FUNCTION_BLOCK L5_Panel
VAR_INPUT
	dr								: REFERENCE TO L1_Director;

	mdF1Producir					: BOOL := TRUE;
	//mdF6Probar						: BOOL;
	mdF5Funcion						: BOOL;
	mdF4Planta						: BOOL;

	hwAS_AvisadorSonoro		AT %Q*	: BOOL; 
	hwLA_LamparaAlarma		AT %Q*	: BOOL; 
	//hwDPO_DesconectaPO		AT %Q*	: BOOL; 	
	hwLM_LamparaMarcha		AT %Q*	: BOOL;
	hwLS_LamparaStop		AT %Q*	: BOOL;

	swF0_Empezar					: BOOL;
	swF1_Producir					: BOOL := TRUE;
	swF2_Preparar					: BOOL := TRUE;
	swF3_Finalizar					: BOOL := TRUE;
	swF6_Probar						: BOOL;
	
	swF4_Planta						: BOOL; 
	swMensaje						: STRING(255) :='';
END_VAR

VAR
	hwPE_Seta					AT %I*	: BOOL;
	swPE_Seta							: BOOL;
	
	hwPOC_PulsadorReset			AT %I*	: BOOL; // POC Botón azul está pulsado (PO Conectada)
	swPOC_PulsadorReset					: BOOL; 
	
	hwPM_PulsadorMarcha			AT %I*	: BOOL; // PM - Pulsador de marcha (verde)
	swPM_PulsadorMarcha					: BOOL;
	fpPM_PulsadorMarcha					: R_TRIG;
	clPM_PulsadorMarcha					: TON;
	
	
	hwPS_PulsadorStop			AT %I*	: BOOL := TRUE; // PS - Pulsador de parada (rojo)
	swPS_PulsadorStop					: BOOL := TRUE; 
	fnPS_PulsadorStop					: F_TRIG; 
	
	hwSM_SelecAutoManual	 	AT %I*	: BOOL; // SM - Selector modo auto/man
	swSM_SelecAutoManual	 			: BOOL; 	

END_VAR


VAR_OUTPUT
	// consignas del panel, resultado de integrar la información que viene del hardware, el estado GEMMA, los temporizadores y flancos, y la interfaz de usuario		
	swF4_Avanza						: BOOL := FALSE;
 	swF4_Retroc						: BOOL := FALSE;	
	
	swF5_Alimentar					: BOOL;
	fpF5_Alimentar					: R_TRIG;  // cuando se pulsa alimentar hay que quitar cargar
	swF5_Situar						: BOOL;
	swF5_Transferir					: BOOL;
	fpF5_Transferir					: R_TRIG; // cuando se pulsa transferir hay que quitar descargar
	swF5_Cargar						: BOOL;
	fpF5_Cargar						: R_TRIG; // cuando se pulsa cargar hay que quitar girar y alimentar
	swF5_Evacuar					: BOOL;
	fpF5_Evacuar					: R_TRIG; // cuando se pulsa evacuar hay que quitar girar
	swF5_Descargar					: BOOL;
	fpF5_Descargar					: R_TRIG; // cuando se pulsa descargar hay que quitar girar y transferir
	swF5_Medir						: BOOL;
	fpF5_Medir						: R_TRIG; // cuano se pulsa medir hay que quitar girar
	swF5_Claridad					: BOOL;
	swF5_Material					: BOOL;
	swF5_Girar						: BOOL;
	fpF5_Girar						: R_TRIG; // cuando se pulsa girar hay que quitar medir, cargar, descargar y evacuar
	swF5_Ejecutar					: BOOL;
	swF5_Ack						: BOOL;
	
END_VAR

VAR
	gmModeName		: STRING 	:= 'Mode A6';
	gmModeDescr		: STRING 	:= 'Inicializando';	
	
//	ttPE_Seta						: STRING := '';

	swA2_FinCiclo					: BOOL;
	swA3_Estado						: BOOL;
	swA6_Inicializar				: BOOL;

	//swF2_Preparar					: BOOL;
	//swF3_Finalizar				: BOOL;	
	//ttF4_Planta						: STRING :='';
	//enF6_Probar						: BOOL;
	//swF6_Probar						: BOOL;
END_VAR

METHOD ProcessCycle : BOOL
VAR_INPUT
	dr				: REFEREnce to L1_Director;
	gmModeActual	: L1_GEMMA;
	tmReinicio 		: TIME; // = dr.tmTiempoReinicio
END_VAR
clPM_PulsadorMarcha(IN:=hwPM_PulsadorMarcha OR  swPM_PulsadorMarcha, PT:=T#1S);
fpPM_PulsadorMarcha(CLK:=hwPM_PulsadorMarcha OR  swPM_PulsadorMarcha);
fnPS_PulsadorStop  (CLK:=hwPS_PulsadorStop   AND swPS_PulsadorStop);

IF hwPE_Seta OR swPE_Seta THEN
	dr.cnD1_Emergencia 				:= TRUE;
	dr.cnA6_Inicializar 			:= FALSE;
	dr.cnA3_Estado					:= FALSE; 
	dr.cnF0_Empezar					:= FALSE;
	dr.cnF4_Planta					:= FALSE; // CON LA SETA NO SE PUEDE ENTRAR EN MODO F4
	dr.cnF5_Funcion					:= FALSE; // CON LA SETA NO SE PUEDE ENTRAR EN MODO F5
	swMensaje 						:= 'Parada de emergencia. Desactive la seta y pulse Reset';

ELSIF dr.cnD1_Emergencia AND NOT (hwPE_Seta OR swPE_Seta) THEN	
	dr.cnD1_Emergencia 				:= FALSE;
	dr.cnA6_Inicializar 			:= TRUE;
	swMensaje 						:= 'Inicializando...';

ELSIF dr.cnA6_Inicializar AND dr.IC THEN
	dr.cnA6_Inicializar				:= FALSE;

ELSIF clPM_PulsadorMarcha.Q THEN			// 1o salta el empezar, si tardas más de 1s luego salta la parada
	dr.cnA3_Estado					:= TRUE;
	dr.cnF0_Empezar					:= FALSE;
	
ELSIF dr.cnF1_Producir AND fnPS_PulsadorStop.Q THEN
	dr.cnA2_FinCiclo				:= TRUE;
	
ELSIF dr.cnA3_Estado AND dr.gmModeActual=L1_GEMMA.A4ParadaObtenida THEN
	dr.cnA3_Estado 					:= FALSE;

ELSIF fpPM_PulsadorMarcha.Q THEN
	dr.cnF0_Empezar 				:= TRUE;
	
ELSIF gmModeActual=L1_GEMMA.A1ParadaInicial THEN
	dr.cnF1_Producir			:= swF1_Producir AND NOT swF6_Probar;
	dr.cnF2_Preparar 			:= swF2_Preparar AND NOT swF6_Probar;
	dr.cnF3_Finalizar			:= swF3_Finalizar AND NOT swF6_Probar;
	dr.cnF6_Probar				:= swF6_Probar AND NOT (swF1_Producir OR swF2_Preparar OR swF3_Finalizar);

ELSIF mdF1Producir AND NOT dr.cnF1_Producir THEN								
	mdF1Producir				:= TRUE;
	mdF4Planta					:= FALSE;
	mdF5Funcion					:= FALSE;
	dr.cnF1_Producir			:= TRUE;
	dr.cnF4_Planta				:= FALSE;	
	dr.cnF5_Funcion				:= FALSE;
	swMensaje					:= 'Modo producción activado';
			
//	dr.cnF1_Producir			:= swF1_Producir AND NOT swF6_Probar;
	//dr.cnF2_Preparar 			:= swF2_Preparar AND NOT swF6_Probar;
	//dr.cnF3_Finalizar			:= swF3_Finalizar AND NOT swF6_Probar;
	//dr.cnF6_Probar				:= swF6_Probar AND NOT (swF1_Producir OR swF2_Preparar OR swF3_Finalizar);		

ELSIF (hwSM_SelecAutoManual OR swSM_SelecAutoManual) AND NOT DR.cnF4_Planta THEN // paso al modo F4
	mdF1Producir				:= FALSE;
	mdF4Planta					:= TRUE;
	mdF5Funcion					:= FALSE;
	dr.cnF1_Producir			:= FALSE;
	dr.cnF4_Planta				:= TRUE;	
	dr.cnF5_Funcion				:= FALSE;
	swMensaje					:= 'Modo mando directo activado';

ELSIF gmModeActual=L1_GEMMA.F4VerificacionSinOrden AND 
	NOT (hwSM_SelecAutoManual OR swSM_SelecAutoManual) THEN
	dr.cnF4_Planta				:= FALSE;
	swSM_SelecAutoManual		:= FALSE;
	swMensaje					:= 'Modo F4 desactivado';

ELSIF mdF5Funcion AND NOT dr.cnF5_Funcion THEN
	mdF1Producir				:= FALSE;
	mdF4Planta					:= FALSE;
	mdF5Funcion					:= TRUE;
	dr.cnF1_Producir			:= FALSE;
	dr.cnF4_Planta				:= FALSE;	
	dr.cnF5_Funcion				:= TRUE;
	swMensaje					:= 'Modo función activado';

END_IF
            




IF gmModeActual=L1_GEMMA.F5VerificacionOrdenada THEN
	
	//IF NOT mdF5Funcion OR NOT mdF5Funcion OR hwSM_SelecAutoManual OR swSM_SelecAutoManual THEN
	//	dr.cnF5_Funcion				:= FALSE;
	//	mdF5Funcion					:= FALSE;
	//	IF hwSM_SelecAutoManual OR swSM_SelecAutoManual THEN
	//		dr.cnF4_Planta			:= TRUE;
	//		swMensaje					:= 'Modo F4 activado';
	//	ELSE
		//	swMensaje					:= 'Modo F5 desactivado';			
		//END_IF
		
	//ELSE
	fpF5_Alimentar				(CLK := swF5_Alimentar);
	fpF5_Cargar					(CLK := swF5_Cargar);
	fpF5_Medir					(CLK := swF5_Medir);
	fpF5_Evacuar				(CLK := swF5_Evacuar);
	fpF5_Descargar				(CLK := swF5_Descargar);
	fpF5_Girar					(CLK :=swF5_Girar);
	fpF5_Transferir				(CLK :=swF5_Transferir);
	IF fpF5_Alimentar.Q AND swF5_Cargar THEN
		swF5_Cargar				:= FALSE; 
		swMensaje				:= 'No se puede cargar si se alimenta';
	ELSIF fpF5_Cargar.Q AND (swF5_Alimentar OR swF5_Girar)THEN
		swF5_Alimentar			:= FALSE; 
		swF5_Girar				:= FALSE;
		swMensaje				:= 'No se puede alimentar ni girar si se carga';		
	ELSIF fpF5_Medir.Q AND swF5_Girar THEN
		swF5_Girar				:= FALSE; 
		swMensaje				:= 'No se puede girar si se mide';
	ELSIF fpF5_Evacuar.Q AND swF5_Girar THEN	
		swF5_Girar				:= FALSE; 
		swMensaje				:= 'No se puede girar si se evacúa';
	ELSIF fpF5_Descargar.Q AND (swF5_Girar OR swF5_Transferir) THEN
		swF5_Girar				:= FALSE; 
		swF5_Transferir			:= FALSE;
		swMensaje				:= 'No se puede girar ni transferir si se descarga';
	ELSIF fpF5_Girar.Q AND (swF5_Cargar OR swF5_Medir OR swF5_Evacuar OR swF5_Descargar) THEN
		swF5_Cargar				:= FALSE;
		swF5_Medir				:= FALSE;
		swF5_Evacuar			:= FALSE;
		swF5_Descargar			:= FALSE;
		swMensaje				:= 'No se puede cargar, medir, evacuar ni descargar si se gira';
	ELSIF fpF5_Transferir.Q AND swF5_Descargar THEN
		swF5_Descargar			:= FALSE; 
		swMensaje				:= 'No se puede descargar si se transfiere';
	END_IF		
END_IF
UpdateUI(gmMode := dr.gmModeActual);

 
//ELSE
	(*

ttPE_Seta := 'Pulsar la seta o el botón para parada de emergencia';	
ttF4_Planta := 'Mandos directos desactivados';
FP_PM(CLk := hwPM_PulsadorMarcha);

dr.cnA1_ParadaIni := FALSE;
	dr.cnA6_Inicializar := FALSE; 
	dr.cnF4_Planta 		:= FALSE;
	dr.cnF5_Funcion 	:= FALSE;
	dr.cnF6_Probar 		:= FALSE;
	dr.cnF1_Producir	:= FALSE;

//----------------------------------------------------------------- Consiga cnD1_Emergencia
dr.cnD1_Emergencia := hwPE_Seta OR swPE_Seta; 
IF dr.cnD1_Emergencia THEN
	IF hwPE_Seta THEN
		IF swPE_Seta THEN
			ttPE_Seta := 'Desarmar la seta y desactivar el botón para reinicializar';
		ELSE
			ttPE_Seta := 'Desarmar la seta para reinicializar';		
		END_IF
	ELSE
		IF swPE_Seta THEN
			ttPE_Seta := 'Desactivar el botón para reinicializar';
		END_IF
	END_IF

//----------------------------------------------------------------- Consigna A6_Inicializar
ELSIF swA6_Inicializar THEN //  OR TmpReinicio.Q);
	// TmpReinicio(IN := hwPM_PulsadorMarcha AND NOT hwPS_PulsadorStop, PT:= tmReinicio);
	dr.cnA6_Inicializar := TRUE; 
	//mdF1Producir := FALSE;
	//mdF4Planta := FALSE;
	//mdF5Funcion := FALSE;
	//mdF6Probar := FALSE;
 
	
//----------------------------------------------------------------- Modo F4_Planta
ELSIF (hwSM_SelecAutoManual OR mdF4Planta) THEN 
	//mdF1Producir 	:= FALSE;
	dr.cnF4_Planta 	:= TRUE;
	//dr.cnF5_Funcion := TRUE;
	//mdF5Funcion 	:= FALSE;
	//mdF6Probar 		:= FALSE;
	IF hwSM_SelecAutoManual AND swF4_Planta THEN
		ttF4_Planta := 'Mandos directos ativados desde panel físico y visualización';
	ELSIF hwSM_SelecAutoManual THEN	
		ttF4_Planta := 'Mandos directos ativados desde panel físico';
	ELSIF swF4_Planta THEN
		ttF4_Planta := 'Mandos directos ativados desde visualización';
	END_IF	

	
	

//----------------------------------------------------------------- F5_Funcion
ELSIF mdF5Funcion THEN  
	//mdF1Producir 	:= FALSE;
	//mdF4Planta 		:= FALSE;
	dr.cnF5_Funcion := TRUE;
	//mdF6Probar 		:= FALSE;

	IF swF5_Girar AND (swF5_Cargar OR swF5_Evacuar OR swF5_Descargar OR swF5_Medir) THEN 
		//swF5_Girar := FALSE;
		swF5_Cargar := FALSE;
		swF5_Evacuar := FALSE;
		swF5_Descargar := FALSE;
		swF5_Medir := FALSE;
		swMensaje := 'No se puede girar a la vez que cargar, evacuar, descargar o medir por riesgo de avería';
	END_IF
	IF swF5_Alimentar AND swF5_Cargar THEN // funciones incompatibles
		swF5_Cargar := FALSE;
		swMensaje := 'No se puede cargar a la vez que alimentar por riesgo de avería';
	END_IF
	IF swF5_Transferir AND swF5_Descargar THEN
		swF5_Transferir := FALSE;
		swMensaje := 'No se puede descargar a la vez que transferer por riesgo de avería';
	END_IF


	
//----------------------------------------------------------------- F6_Probar
ELSIF mdF6Probar THEN  
	//mdF1Producir	:= FALSE;
	//mdF4Planta 		:= FALSE;
	//mdF5Funcion 	:= FALSE;
	dr.cnA1_ParadaIni := NOT dr.cnF0_Empezar;
	dr.cnF6_Probar 	:= TRUE;
	IF (swF0_Empezar OR FP_PM.Q) THEN
		dr.cnF0_Empezar := TRUE;
	END_IF

	
//----------------------------------------------------------------- F1_Producir
ELSIF (mdF1Producir OR FP_PM.Q) THEN
	dr.cnF1_Producir:= TRUE;

	IF (swF0_Empezar OR FP_PM.Q) THEN
		dr.cnF0_Empezar := TRUE;
	END_IF
	//dr.cnF0_Empezar := (swF0_Empezar OR FP_PM.Q);  
	dr.cnA1_ParadaIni := NOT dr.cnF0_Empezar;
	//mdF4Planta 		:= FALSE;
	//mdF5Funcion 	:= FALSE;
	//mdF6Probar	 	:= FALSE;

	dr.cnA2_FinCiclo:= (swA2_FinCiclo OR hwPS_PulsadorStop); // enA2_FinCiclo AND (swA2_FinCiclo OR hwPS_PulsadorStop);
	dr.cnA3_Estado 	:= swA3_Estado;

ELSE
	dr.cnF0_Empezar :=FALSE; 
	//dr.cnA1_ParadaIni 	:= TRUE;
	dr.cnA6_Inicializar := FALSE; 
	dr.cnF4_Planta 		:= FALSE;
	dr.cnF5_Funcion 	:= FALSE;
	dr.cnF6_Probar 		:= FALSE;
	dr.cnF1_Producir	:= FALSE;
END_IF 

IF dr.Failure OR dr.gmModeActual=L1_GEMMA.A4ParadaObtenida OR dr.gmModeActual=L1_GEMMA.D2TratamientoFallos THEN
	dr.cnF0_Empezar := FALSE;
	IF (swF0_Empezar OR FP_PM.Q) THEN
		dr.cnF0_Empezar := TRUE;
	END_IF	
END_IF

(*
dr.cnF1_Empezar := enF1_Empezar AND (swF1_Empezar OR FP_PM.Q);
IF NOT dr.cnF1_Empezar AND (swF1_Empezar OR FP_PM.Q) THEN // consigna no válida
	swF1_Empezar := FALSE; // si no se puede entrar en el modo hay que desactivar el botón
	swMensaje := 'Sólo se puede empezar desde una parada';
END_IF

//----------------------------------------------------------------- Consigna A2_ParaFinCiclo

IF NOT dr.cnA2_FinCiclo AND (swA2_FinCiclo OR hwPS_PulsadorStop) THEN // consigna no válida
	swA2_FinCiclo := FALSE; // si no se puede entrar en el modo hay que desactivar el botón
	swMensaje := 'Sólo se puede pasar a A2 desde el modo F1';

ELS 
IF dr.cnA2_FinCiclo THEN
	// swA2_FinCiclo := TRUE; 
	IF gmModeActual = L1_GEMMA.F1ProduccionNormal THEN
		swMensaje := 'Esperando a finalizar el ciclo para parar';
	ELSIF gmModeActual = L1_GEMMA.A4ParadaObtenida THEN
		swMensaje := 'Parada obtenida después de acabar el ciclo';
	END_IF
END_IF 
dr.cnA3_Estado := enA3_Estado AND (swA3_Estado);
IF NOT dr.cnA3_Estado AND (swA3_Estado) THEN // consigna no válida
	swA3_Estado := FALSE; // si no se puede entrar en el modo hay que desactivar el botón
	swMensaje := 'Sólo se puede pasar a A3 desde el modo F1, F5 o A2';

ELSIF dr.cnA3_Estado THEN
	swA3_Estado := TRUE; 
	IF gmModeActual = L1_GEMMA.A4ParadaObtenida THEN
		swMensaje := 'Parada obtenida después de alcanzar un estado estable';
	ELSE
		swMensaje := 'Esperando a un estado estable para parar';
	END_IF
END_IF

//----------------------------------------------------------------- Consigna F1_Reanudar
dr.cnF1_Reanudar := enF1_Reanduar AND (swF1_Reanudar OR hwPM_PulsadorMarcha);
 	
IF NOT dr.cnF1_Reanudar AND (swF1_Reanudar OR hwPM_PulsadorMarcha) THEN // consigna no válida
	swF1_Reanudar := FALSE; // si no se puede entrar en el modo hay que desactivar el botón
	swMensaje := 'Sólo se puede reanudar desde una parada';

ELSIF dr.cnF1_Reanudar THEN
	swMensaje := 'Reanundando tras la parada';
END_IF

//----------------------------------------------------------------- Consigna A3_Estado
	
*)







*)

//----------------------------------------------------------------- Consigna F1_Empezar

//END_IF
END_METHOD

METHOD UpdateUi : BOOL
VAR_INPUT
	gmMode				: L1_GEMMA;
END_VAR
// actualizar actuadores del panel
hwAS_AvisadorSonoro 			:= FALSE;
hwLA_LamparaAlarma				:= FALSE;
hwLM_LamparaMarcha				:= FALSE;

CASE gmMode OF
	L1_GEMMA.A1ParadaInicial:
		gmModeName				:= 'Mode A1';
		gmModeDescr				:= 'Parada en estado inicial';
		hwLM_LamparaMarcha		:= dr.Tic;
		
	L1_GEMMA.A2ParaFinCiclo:
		gmModeName				:= 'Mode A2';
		gmModeDescr				:= 'Parada a final de ciclo solicitada';
		hwLM_LamparaMarcha		:= TRUE;
		
	L1_GEMMA.A3ParadaEstado:
		gmModeName				:= 'Mode A3';
		gmModeDescr				:= 'Parada en estado actual solicitada';
		
	L1_GEMMA.A4ParadaObtenida:
		gmModeName				:= 'Mode A4';
		gmModeDescr				:= 'Parada obtenida';
		hwLM_LamparaMarcha		:= dr.Tic;
		
	L1_GEMMA.A5PreparandoTrasFallo:
		gmModeName				:= 'Mode A5';
		gmModeDescr				:= 'Preparando tras fallo';	
		
	L1_GEMMA.A6Inicializando:
		gmModeName				:= 'Mode A6';
		gmModeDescr				:= 'Inicializando';
		hwLA_LamparaAlarma		:= dr.Tic;
		//hwDPO_DesconectaPO		:= dr.Tic;
		
	L1_GEMMA.A7SituandoEstado:
		gmModeName				:= 'Mode A7';
		gmModeDescr				:= 'Situando PO en un estado determinado';

	L1_GEMMA.F1ProduccionNormal:
		gmModeName				:= 'Mode F1';
		gmModeDescr				:= 'Producción normal';
		hwLM_LamparaMarcha		:= TRUE;

	L1_GEMMA.F2SecuenciaPreparacion:
		gmModeName				:= 'Mode F2';
		gmModeDescr				:= 'Secuencia de preparación';	
		hwAS_AvisadorSonoro 	:= dr.Tic;
		hwLM_LamparaMarcha		:= TRUE;
		
	L1_GEMMA.F3SecuenciaFinalizacion:
		gmModeName				:= 'Mode F3';
		gmModeDescr				:= 'Secuencia de finalización';
		hwAS_AvisadorSonoro 	:= TRUE;
		hwLM_LamparaMarcha		:= TRUE;
		
	L1_GEMMA.F4VerificacionSinOrden:
		gmModeName				:= 'Mode F4';
		gmModeDescr				:= 'Verificación sin orden (Planta)';
		
	L1_GEMMA.F5VerificacionOrdenada:
		gmModeName				:= 'Mode F5';
		gmModeDescr				:= 'Verificación ordenada (Función)';
				
	L1_GEMMA.F6Probando:
		gmModeName				:= 'Mode F6';
		gmModeDescr				:= 'Probando';
		
	L1_GEMMA.D1ParadaEmergencia:
		gmModeName				:= 'Mode D1';
		gmModeDescr				:= 'Parada de emergencia';
		hwAS_AvisadorSonoro 	:= dr.Tic;
		hwLA_LamparaAlarma		:= dr.Tic;

	L1_GEMMA.D2TratamientoFallos:
		gmModeName				:= 'Mode D2';
		gmModeDescr				:= 'Diagnósdr.tico/tratamiento de fallos';
		hwAS_AvisadorSonoro 	:= dr.Tic;
		hwLA_LamparaAlarma		:= dr.Tic;
		
	L1_GEMMA.D3ProducirConFallos:
		gmModeName				:= 'Mode D3';
		gmModeDescr				:= 'Producir con fallos';

END_CASE
END_METHOD

END_FUNCTION_BLOCK

(* stored: Version 1.1.0.1, ProductVersion 3.1.4024.11
   POU L5_Panel: Id {514e5db3-ac71-4add-977b-df9fa295436c}, SpecialFunc None
   Method ProcessCycle: Id {026a1e81-704d-4f95-ae3e-7d143e02920e}
   Method UpdateUi: Id {2f7a7a64-69c4-4b55-9d9b-f8c62855d55d} *)
